(* PLC project SafeLOGIC, BrAutomation SafeDESIGNER  5.24.1.0 *)
(* stored: companyURL http://www.br-automation.com, creationDateTime Fri Nov 28 15:29:43 2025 *)

PROGRAM Main
  VAR  (* added by the conversion: wires and edge detectors of the diagram *)
    _MUL_S5_OUT : SAFEINT;
    _GE_S113_OUT : SAFEDINT;
    _AND_S145_OUT : SAFEINT;
    _NOT_S51_OUT : BOOL;
    _OR_S127_OUT : ANY;
  END_VAR

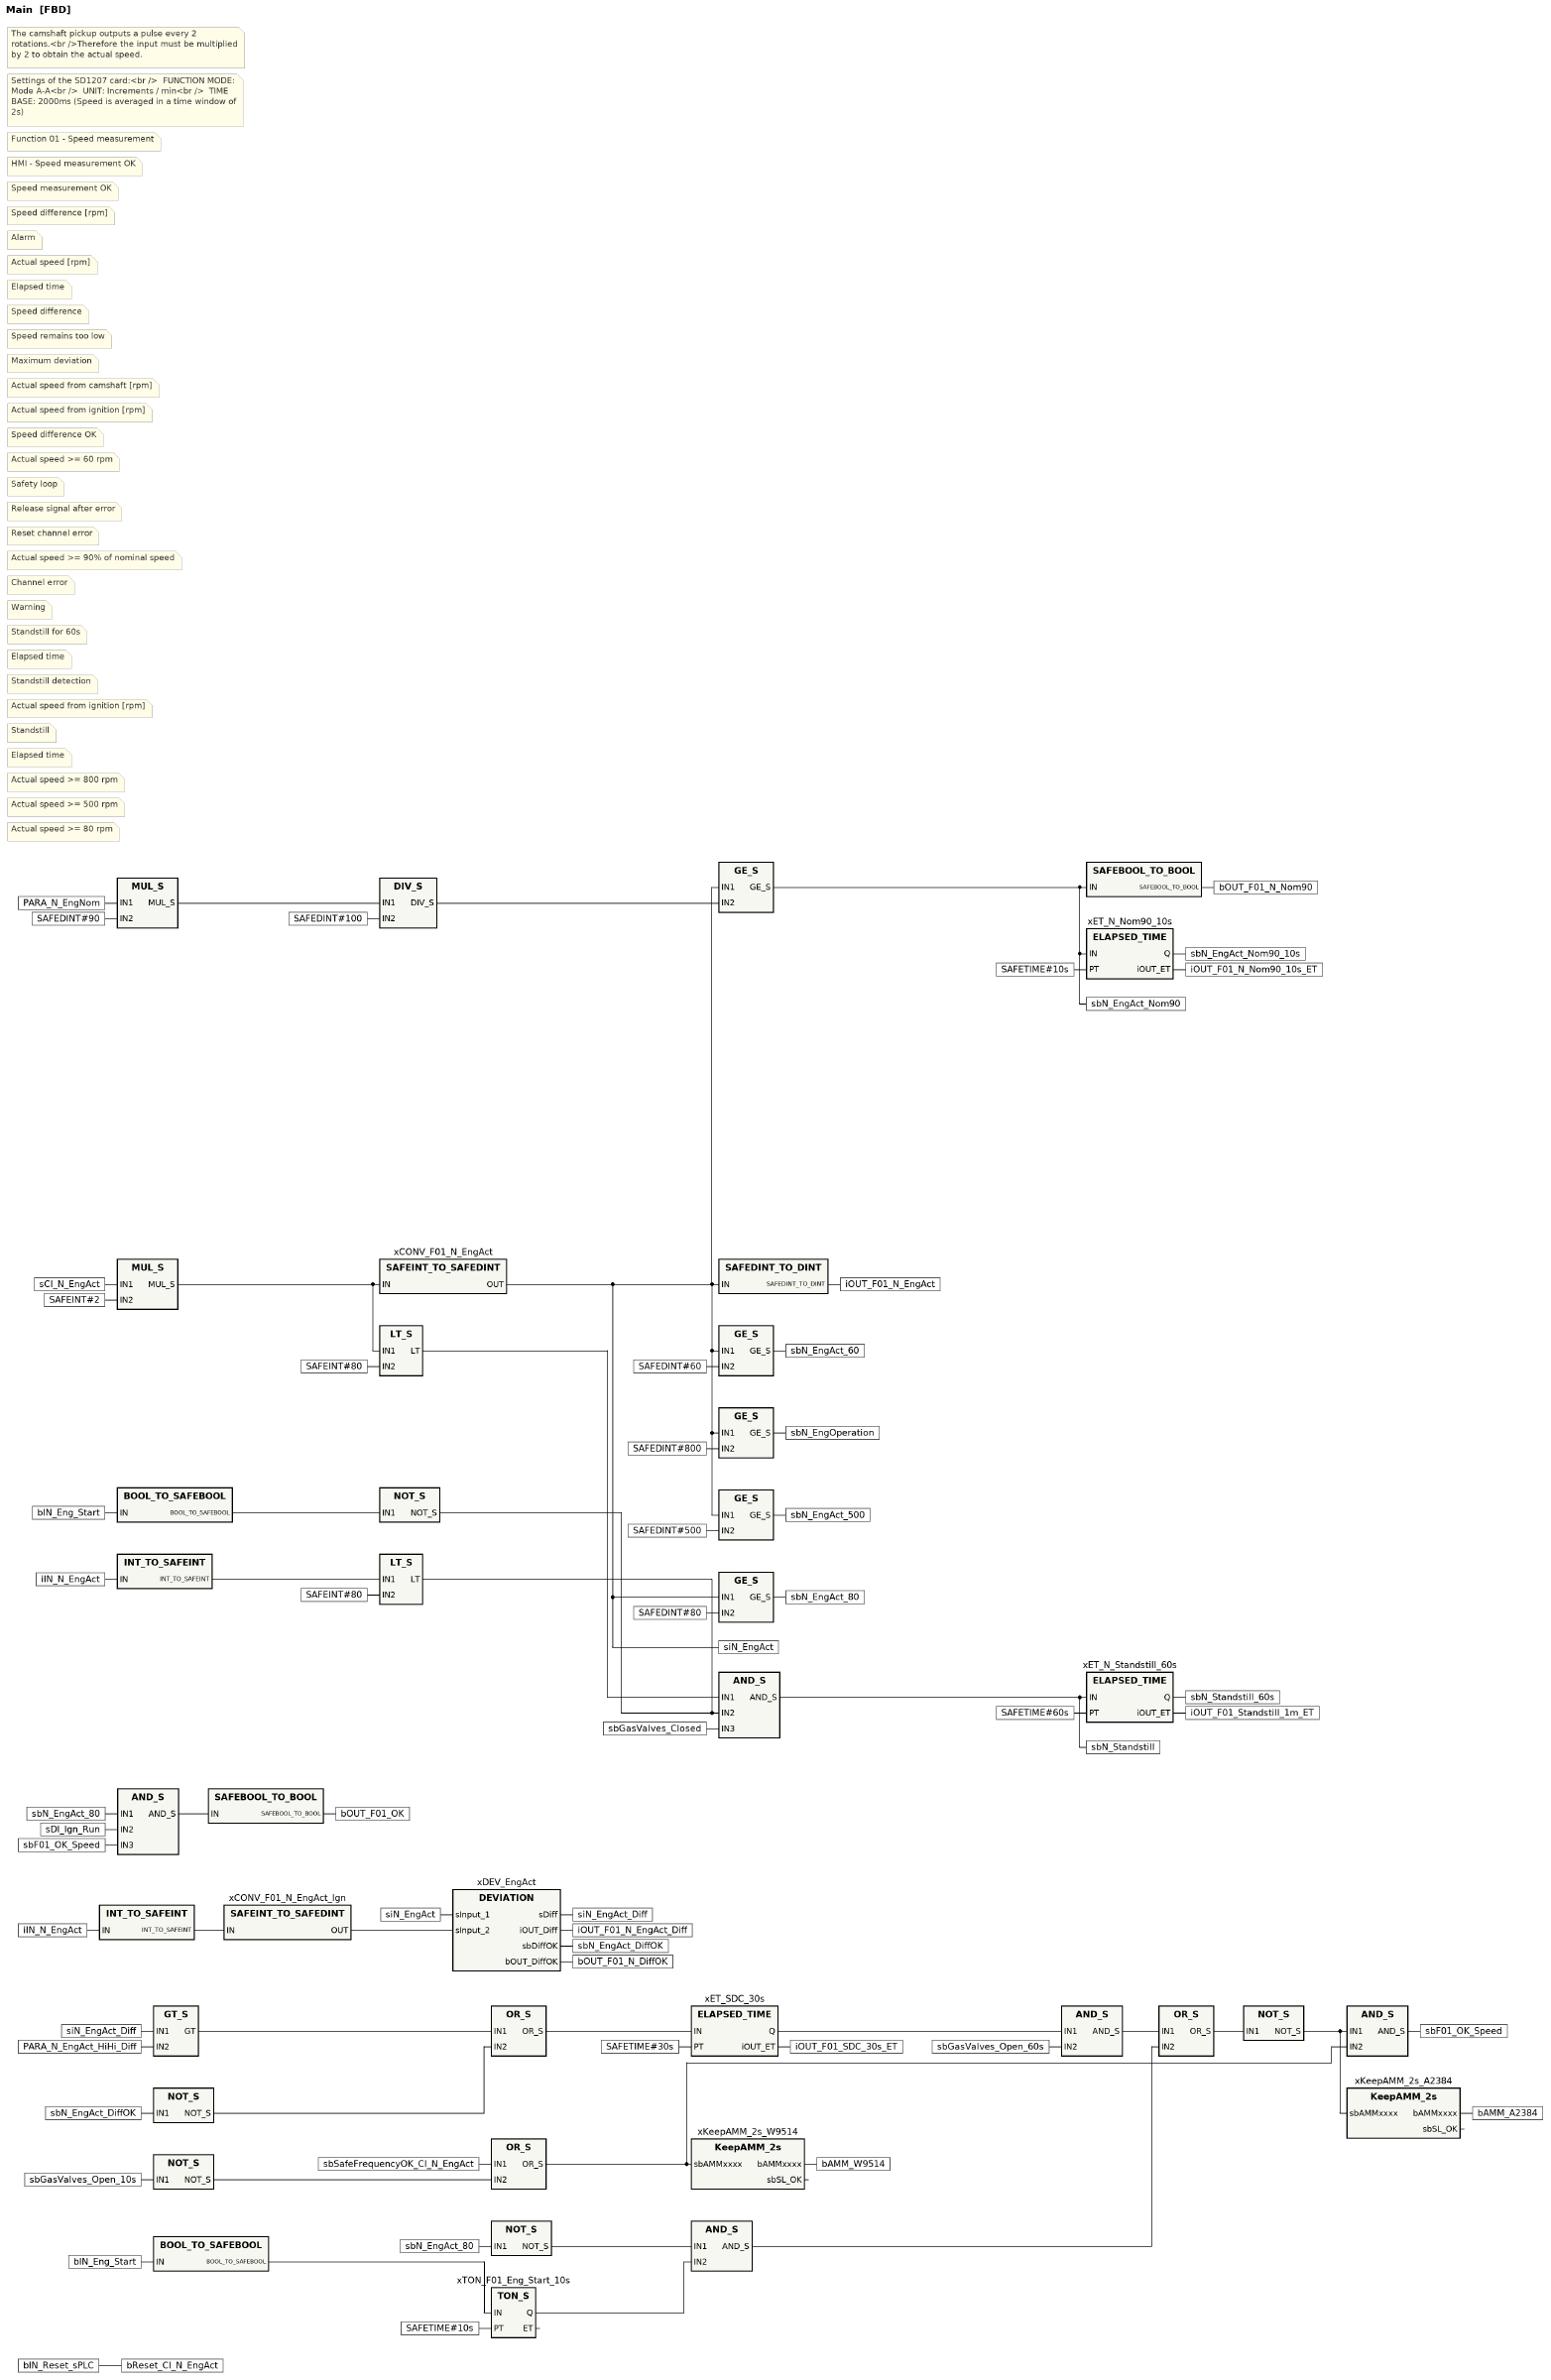
(* FBD diagram, written out as Structured Text *)
(* Function 01 - Speed measurement *)
(* Settings of the SD1207 card:<br />  FUNCTION MODE: Mode A-A<br />  UNIT: Increments / min<br />  TIME BASE: 2000ms (Speed is averaged in a time window of 2s) *)
(* The camshaft pickup outputs a pulse every 2 rotations.<br />Therefore the input must be multiplied by 2 to obtain the actual speed. *)
(* Actual speed [rpm] *)
_MUL_S5_OUT := MUL_S(sCI_N_EngAct, SAFEINT#2);
xCONV_F01_N_EngAct(IN := _MUL_S5_OUT);
siN_EngAct := xCONV_F01_N_EngAct.OUT;
(* Actual speed >= 60 rpm *)
iOUT_F01_N_EngAct := SAFEDINT_TO_DINT(xCONV_F01_N_EngAct.OUT);
sbN_EngAct_60 := GE_S(xCONV_F01_N_EngAct.OUT, SAFEDINT#60);
(* Actual speed >= 80 rpm *)
(* Actual speed >= 500 rpm *)
(* Actual speed >= 800 rpm *)
(* Actual speed >= 90% of nominal speed *)
_GE_S113_OUT := GE_S(xCONV_F01_N_EngAct.OUT, DIV_S(MUL_S(PARA_N_EngNom, SAFEDINT#90), SAFEDINT#100));
sbN_EngAct_Nom90 := _GE_S113_OUT;
sbN_EngOperation := GE_S(xCONV_F01_N_EngAct.OUT, SAFEDINT#800);
sbN_EngAct_500 := GE_S(xCONV_F01_N_EngAct.OUT, SAFEDINT#500);
sbN_EngAct_80 := GE_S(xCONV_F01_N_EngAct.OUT, SAFEDINT#80);
(* Elapsed time *)
xET_N_Nom90_10s(IN := _GE_S113_OUT, PT := SAFETIME#10s);
sbN_EngAct_Nom90_10s := xET_N_Nom90_10s.Q;
bOUT_F01_N_Nom90 := SAFEBOOL_TO_BOOL(_GE_S113_OUT);
iOUT_F01_N_Nom90_10s_ET := xET_N_Nom90_10s.iOUT_ET;
(* Standstill detection *)
(* Standstill *)
(* Actual speed from ignition [rpm] *)
(* Standstill for 60s *)
(* Elapsed time *)
_AND_S145_OUT := AND_S(LT_S(_MUL_S5_OUT, SAFEINT#80), LT_S(INT_TO_SAFEINT(iIN_N_EngAct), SAFEINT#80), NOT_S(BOOL_TO_SAFEBOOL(bIN_Eng_Start)), sbGasValves_Closed);
xET_N_Standstill_60s(IN := _AND_S145_OUT, PT := SAFETIME#60s);
sbN_Standstill_60s := xET_N_Standstill_60s.Q;
sbN_Standstill := _AND_S145_OUT;
iOUT_F01_Standstill_1m_ET := xET_N_Standstill_60s.iOUT_ET;
(* Speed difference *)
(* Actual speed from camshaft [rpm] *)
(* Speed difference [rpm] *)
(* Actual speed from ignition [rpm] *)
xCONV_F01_N_EngAct_Ign(IN := INT_TO_SAFEINT(iIN_N_EngAct));
xDEV_EngAct(sInput_1 := siN_EngAct, sInput_2 := xCONV_F01_N_EngAct_Ign.OUT);
iOUT_F01_N_EngAct_Diff := xDEV_EngAct.iOUT_Diff;
(* Speed difference OK *)
sbN_EngAct_DiffOK := xDEV_EngAct.sbDiffOK;
siN_EngAct_Diff := xDEV_EngAct.sDiff;
bOUT_F01_N_DiffOK := xDEV_EngAct.bOUT_DiffOK;
(* Maximum deviation *)
(* Alarm *)
xET_SDC_30s(IN := OR_S(GT_S(siN_EngAct_Diff, PARA_N_EngAct_HiHi_Diff), NOT_S(sbN_EngAct_DiffOK)), PT := SAFETIME#30s);
xTON_F01_Eng_Start_10s(IN := BOOL_TO_SAFEBOOL(bIN_Eng_Start), PT := SAFETIME#10s);
_NOT_S51_OUT := NOT_S(OR_S(AND_S(xET_SDC_30s.Q, sbGasValves_Open_60s), AND_S(NOT_S(sbN_EngAct_80), xTON_F01_Eng_Start_10s.Q)));
xKeepAMM_2s_A2384(sbAMMxxxx := _NOT_S51_OUT);
bAMM_A2384 := xKeepAMM_2s_A2384.bAMMxxxx;
(* Elapsed time *)
(* Safety loop *)
iOUT_F01_SDC_30s_ET := xET_SDC_30s.iOUT_ET;
_OR_S127_OUT := OR_S(sbSafeFrequencyOK_CI_N_EngAct, NOT_S(sbGasValves_Open_10s));
sbF01_OK_Speed := AND_S(_NOT_S51_OUT, _OR_S127_OUT);
(* Speed remains too low *)
(* Channel error *)
(* Warning *)
xKeepAMM_2s_W9514(sbAMMxxxx := _OR_S127_OUT);
bAMM_W9514 := xKeepAMM_2s_W9514.bAMMxxxx;
(* HMI - Speed measurement OK *)
(* Speed measurement OK *)
bOUT_F01_OK := SAFEBOOL_TO_BOOL(AND_S(sbN_EngAct_80, sDI_Ign_Run, sbF01_OK_Speed));
(* Release signal after error *)
(* Reset channel error *)
bReset_CI_N_EngAct := bIN_Reset_sPLC;
END_PROGRAM
